FUNCTION_BLOCK FB_WeightHistory
VAR_INPUT
    eWeight1RunningState : INT;
    eWeight2RunningState : INT;
    eWeight3RunningState : INT;
    eWeight4RunningState : INT;

    WeightMeasured_1      : LREAL;
    CorrectionWeight_1    : LREAL;
    WeightMeasured_2      : LREAL;
    CorrectionWeight_2    : LREAL;
    WeightMeasured_3      : LREAL;
    CorrectionWeight_3    : LREAL;
    WeightMeasured_4      : LREAL;
    CorrectionWeight_4    : LREAL;
END_VAR

VAR_IN_OUT
    aWeightPoints : ARRAY [0..7,0..9999] OF ST_Point_1;
END_VAR

VAR
    fbTrig1 : R_TRIG;
    fbTrig2 : R_TRIG;
    fbTrig3 : R_TRIG;
    fbTrig4 : R_TRIG;

	fileTime : T_FILETIME64;
    dtNow    : DT;

    i           : INT;
END_VAR

// ----------------------------------------
// 1) Pobierz aktualny czas systemowy (FILETIME64)
// ----------------------------------------
fileTime := F_GetSystemTime();

// ----------------------------------------
// 2) FILETIME64 → DT (pełna data i czas)
// ----------------------------------------
dtNow := FILETIME64_TO_DT(fileTime);




// --------------------------	
// WAGA 1
// --------------------------
fbTrig1(CLK := (eWeight1RunningState = 3));   // flanka na stanie 3
IF fbTrig1.Q THEN
    // kolumna 0: WeightMeasured
    FOR i := 0 TO 9998 DO
        aWeightPoints[0, i] := aWeightPoints[0, i + 1];
    END_FOR
    aWeightPoints[0, 9999].x := dtNow;
    aWeightPoints[0, 9999].y := LREAL_TO_INT(WeightMeasured_1);

    // kolumna 1: CorrectionWeight
    FOR i := 0 TO 9998 DO
        aWeightPoints[4, i] := aWeightPoints[4, i + 1];
    END_FOR
    aWeightPoints[4, 9999].x := dtNow;
    aWeightPoints[4, 9999].y := LREAL_TO_INT(CorrectionWeight_1);
END_IF


// --------------------------
// WAGA 2
// --------------------------
fbTrig2(CLK := (eWeight2RunningState = 3));
IF fbTrig2.Q THEN
    // kolumna 2: WeightMeasured
    FOR i := 0 TO 9998 DO
        aWeightPoints[1, i] := aWeightPoints[1, i + 1];
    END_FOR
    aWeightPoints[1, 9999].x := dtNow;
    aWeightPoints[1, 9999].y := LREAL_TO_INT(WeightMeasured_2);

    // kolumna 3: CorrectionWeight
    FOR i := 0 TO 9998 DO
        aWeightPoints[5, i] := aWeightPoints[5, i + 1];
    END_FOR
    aWeightPoints[5, 9999].x := dtNow;
    aWeightPoints[5, 9999].y := LREAL_TO_INT(CorrectionWeight_2);
END_IF


// --------------------------
// WAGA 3
// --------------------------
fbTrig3(CLK := (eWeight3RunningState = 3));
IF fbTrig3.Q THEN
    // kolumna 4: WeightMeasured
    FOR i := 0 TO 9998 DO
        aWeightPoints[2, i] := aWeightPoints[2, i + 1];
    END_FOR
    aWeightPoints[2, 9999].x := dtNow;
    aWeightPoints[2, 9999].y := LREAL_TO_INT(WeightMeasured_3);

    // kolumna 5: CorrectionWeight
    FOR i := 0 TO 9998 DO
        aWeightPoints[6, i] := aWeightPoints[6, i + 1];
    END_FOR
    aWeightPoints[6, 9999].x := dtNow;
    aWeightPoints[6, 9999].y := LREAL_TO_INT(CorrectionWeight_3);
END_IF


// --------------------------
// WAGA 4
// --------------------------
// UWAGA: tu według Twojego opisu stan = 4
fbTrig4(CLK := (eWeight4RunningState = 3));
IF fbTrig4.Q THEN
    // kolumna 6: WeightMeasured
    FOR i := 0 TO 9998 DO
        aWeightPoints[3, i] := aWeightPoints[3, i + 1];
    END_FOR
    aWeightPoints[3, 9999].x := dtNow;
    aWeightPoints[3, 9999].y := LREAL_TO_INT(WeightMeasured_4);

    // kolumna 7: CorrectionWeight
    FOR i := 0 TO 9998 DO
        aWeightPoints[7, i] := aWeightPoints[7, i + 1];
    END_FOR
    aWeightPoints[7, 9999].x := dtNow;
    aWeightPoints[7, 9999].y := LREAL_TO_INT(CorrectionWeight_4);
END_IF

END_FUNCTION_BLOCK

(* stored: Version 1.2.0.0, ProductVersion 3.1.4026.13, FileIdentifier a4959769deb15670dd046b67e05ea4d1f28e0dda, FileSignature a4e8f97a6ee1fdfaec5db9fdab1ed704b7e2da1e94c6494b8fd42e48ee2c758e58442aa2f72fc524a065731886906163056c2fe86820d223dc2e96425eb54f5a02324310492148b10c98408de53438a12776dc99bed38a1bfdb8f78e034480c1759313d426bcfb8c685a838efdd6636f1b9613c2b760f56d92d5f983adf532cb52f1c5dc246b182c997d74169b3f0507d5d8547c88979a42bd512c8ac90ab01511b77ef6157cc7b083ac620d903f1803509211876fc2c195ecc52b17f6c586d6ad6b3cf0049a2613a27eda237c576f0386a0188962f56b4f7830b551a8a3fd78bf828d489adb16e0d74f53659385d80a2f11384dc5e3c16e591cb35412b9e51b
   POU FB_WeightHistory: Id {24a1b0f3-4555-43dc-ab97-872bd894b563}, SpecialFunc None *)
